Fanuc KAREL source: NC0076.KL

-- PROVISIONAL review KL for V1013-1; original PC SHA256 cdb797eb96e2ecd1ffc97cc3b9e99ed63ea027337d67104d9a2a36f6806d671a
-- Incomplete behavior may be omitted. Consult companion uncertainty JSON. Do not deploy.
PROGRAM NC0076
%NOLOCKGROUP
-- UNRESOLVED_LOCAL_POOL 1 cells at code offset 3; source declarations unknown
-- DIRECT_LOCAL_WORD_ACCESS alone does not prove INTEGER, REAL, or BOOLEAN
BEGIN
  -- UNRESOLVED_PC offsets 0-8; opcodes 2B,2C,7B
  -- UNRESOLVED_PC offsets 13-20; opcodes 9D,23
  -- UNRESOLVED_PC offsets 25-42; opcodes 21,2E,59,79
  -- UNRESOLVED_PC offsets 47-64; opcodes 21,2E,59,79
  -- UNRESOLVED_PC offsets 69-86; opcodes 21,2E,59,79
  -- UNRESOLVED_PC offsets 91-108; opcodes 21,2E,59,79
  -- UNRESOLVED_PC offsets 113-130; opcodes 21,2E,59,79
  -- UNRESOLVED_PC offsets 135-152; opcodes 21,2E,59,79
  -- UNRESOLVED_PC offsets 157-174; opcodes 21,2E,59,79
  -- UNRESOLVED_PC offsets 179-196; opcodes 21,2E,59,79
  -- UNRESOLVED_PC offsets 201-215; opcodes 21,9D,52,23
  -- UNRESOLVED_PC offsets 220-225; opcodes 7A
  -- UNRESOLVED_PC offsets 230-235; opcodes 7A
  -- UNRESOLVED_PC offsets 240-245; opcodes 7A
  -- UNRESOLVED_PC offsets 250-255; opcodes 7A
  -- UNRESOLVED_PC offsets 260-265; opcodes 7A
  -- UNRESOLVED_PC offsets 270-275; opcodes 7A
  -- UNRESOLVED_PC offsets 280-285; opcodes 7A
  -- UNRESOLVED_PC offsets 290-295; opcodes 7A
  -- UNRESOLVED_PC offsets 300-304; opcodes 7F
  -- UNRESOLVED_PC offsets 309-313; opcodes 27,AA
  -- UNRESOLVED_PC offsets 318-322; opcodes 7F
END NC0076
